(* CoDeSys 2.3 export: TRANSPORTCLASS.EXP *)

(* Data type in ENUM *)
TYPE TransportClass : (Forced:=1, Passive);
END_TYPE
